{attribute 'GeneratedUsingTerminal: EK1122-0000-0018'}
{attribute addProperty BoxType "EK1122-0000-0018"}
{attribute addProperty Id "Beckhoff_ATH2xxxsub_EK1100EK1100_1FC0878B2A_0001_ATH2000_0250_0022A_0001_ATH2000_0250_0022_300D1FD014A_0002_ATH2000_0250_0023A_0002_ATH2000_0250_0023_E62B11EA14A_0003_ATH2000_0250_0024ATH2000_A7FEA1CF76A_0004_ATH2040_0250_0022ATH2040_A7FEA1CF76A_0005_ATH2040_0250_0023ATH2040_A7FEA1CF76A_0006_ATH2040_0250_0024ATH2040_A7FEA1CF76A_0007_ATH2050_0500_0022ATH2050_A7FEA1CF76A_0008_ATH2050_0500_0023ATH2050_A7FEA1CF76A_0009_ATH2050_0500_0024ATH2050_A7FEA1CF76A_0010_ATH2050_0501_0022ATH2050_A7FEA1CF76A_0011_ATH2050_0501_0023ATH2050_A7FEA1CF76A_0012_ATH2050_0501_0024ATH2050_A7FEA1CF76"}
{attribute addProperty CRC "838265480"}
{attribute addProperty Size "790"}
TYPE Beckhoff_ATH2xxxEK1122_31F6EA88 EXTENDS EK1122_1FC0878B :
STRUCT
	{attribute addProperty Name "Beckhoff_ATH2xxxsub_EK1100"}
	{attribute addProperty PreviousPort "Beckhoff ATH2xxxEK1122 : D"}
	Beckhoff_ATH2xxxsub_EK1100 : EK1100_1FC0878B;
	{attribute addProperty Name "A_0001_ATH2000_0250_0022"}
	{attribute addProperty PreviousPort "Beckhoff ATH2xxxsub EK1100 : C"}
	A_0001_ATH2000_0250_0022 : A_0001_ATH2000_0250_0022_300D1FD0;
	{attribute addProperty Name "A_0002_ATH2000_0250_0023"}
	{attribute addProperty PreviousPort "A_0001(ATH2000-0250-0022) : C"}
	A_0002_ATH2000_0250_0023 : A_0002_ATH2000_0250_0023_E62B11EA;
	{attribute addProperty Name "A_0003_ATH2000_0250_0024"}
	{attribute addProperty PreviousPort "A_0002(ATH2000-0250-0023) : C"}
	A_0003_ATH2000_0250_0024 : ATH2000_A7FEA1CF;
	{attribute addProperty Name "A_0004_ATH2040_0250_0022"}
	{attribute addProperty PreviousPort "A_0003(ATH2000-0250-0024) : C"}
	A_0004_ATH2040_0250_0022 : ATH2040_A7FEA1CF;
	{attribute addProperty Name "A_0005_ATH2040_0250_0023"}
	{attribute addProperty PreviousPort "A_0004(ATH2040-0250-0022) : C"}
	A_0005_ATH2040_0250_0023 : ATH2040_A7FEA1CF;
	{attribute addProperty Name "A_0006_ATH2040_0250_0024"}
	{attribute addProperty PreviousPort "A_0005(ATH2040-0250-0023) : C"}
	A_0006_ATH2040_0250_0024 : ATH2040_A7FEA1CF;
	{attribute addProperty Name "A_0007_ATH2050_0500_0022"}
	{attribute addProperty PreviousPort "A_0006(ATH2040-0250-0024) : C"}
	A_0007_ATH2050_0500_0022 : ATH2050_A7FEA1CF;
	{attribute addProperty Name "A_0008_ATH2050_0500_0023"}
	{attribute addProperty PreviousPort "A_0007(ATH2050-0500-0022) : C"}
	A_0008_ATH2050_0500_0023 : ATH2050_A7FEA1CF;
	{attribute addProperty Name "A_0009_ATH2050_0500_0024"}
	{attribute addProperty PreviousPort "A_0008(ATH2050-0500-0023) : C"}
	A_0009_ATH2050_0500_0024 : ATH2050_A7FEA1CF;
	{attribute addProperty Name "A_0010_ATH2050_0501_0022"}
	{attribute addProperty PreviousPort "A_0009(ATH2050-0500-0024) : C"}
	A_0010_ATH2050_0501_0022 : ATH2050_A7FEA1CF;
	{attribute addProperty Name "A_0011_ATH2050_0501_0023"}
	{attribute addProperty PreviousPort "A_0010(ATH2050-0501-0022) : C"}
	A_0011_ATH2050_0501_0023 : ATH2050_A7FEA1CF;
	{attribute addProperty Name "A_0012_ATH2050_0501_0024"}
	{attribute addProperty PreviousPort "A_0011(ATH2050-0501-0023) : C"}
	A_0012_ATH2050_0501_0024 : ATH2050_A7FEA1CF;
END_STRUCT
END_TYPE

(* stored: Version 1.2.0.0, ProductVersion 3.1.4024.9
   DUT Beckhoff_ATH2xxxEK1122_31F6EA88: Id {bb9b3399-1219-4990-8977-6cb72345fdc3} *)
